// TIA Portal V20 program export: 7 tag tables, 9 data types, 98 data blocks, 45 code blocks (in call order from the OBs), 102 instance data blocks

VAR_GLOBAL   // PLC tag table "00_Simulation"
   "AAxxxSP1.Slot1.I.16" AT %I1.0 : Bool;   // SIMIT Simulation currently running (life bit from SIMIT, always TRUE while SIMIT is running)
END_VAR

VAR_GLOBAL   // PLC tag table "06_ProductionData"
END_VAR
VAR_GLOBAL CONSTANT   // user constants
   NO_DATASETS_CYCLETIMER : Int := 8;   // SICAR: Anzahl Datensätze Taktzeiten / SICAR: Number of data sets Cycle Timer
   NO_DATASETS_LIMITVALUES : Int := 2;   // SICAR: Anzahl Datensätze Grenzwerte / SICAR: Number of data sets Limit Value
   NO_DATASETS_SHIFTCOUNTER : Int := 2;   // SICAR: Anzahl Datensätze Schichtzähler / SICAR: Number of data sets Shift Counter
   NO_DATASETS_COUNTER : Int := 2;   // SICAR: Anzahl Datensätze Zähler / SICAR: Number of data sets Counter
END_VAR

VAR_GLOBAL   // PLC tag table "07_Energy"
   PAC3220InPut AT %I500.0 : "LER_typePAC3220ProfinetInput";
   PAC3220OutPut AT %Q500.0 : "LER_typePAC3220ProfinetOutput";
   "Active energy import tariff 1(F)" AT %ID612 : Real;
   "Reactive energy import tariff 1 (F)" AT %ID616 : Real;
   "Apparent energy tariff 1 (F)" AT %ID620 : Real;
   "Active energy export tariff 1(F)" AT %ID624 : Real;
   "Reactive energy export tariff 1 (F)" AT %ID628 : Real;
   "Apparent power L1" AT %ID632 : Real;
   "Apparent power L2" AT %ID636 : Real;
   "Apparent power L3" AT %ID640 : Real;
   "Active power L1" AT %ID644 : Real;
   "Active power L2" AT %ID648 : Real;
   "Active power L3" AT %ID652 : Real;
   "Reactive power L1" AT %ID656 : Real;
   "Reactive power L2" AT %ID660 : Real;
   "Reactive power L3" AT %ID664 : Real;
END_VAR
VAR_GLOBAL CONSTANT   // user constants
   NO_OF_MACHINES : USInt := 1;   // SICAR: No of machines for EE-Monitor
   NO_OF_MEASUREPOINTS : USInt := 1;   // SICAR: Anzahl der Messstellen für EE-Monitor / SICAR: No of measurepoints for EE-Monitor
   "DP_FRWA1_1_0_000CC1-KE50~DP_FRWA1_1_0_000CC1-KE50_900" : Hw_Io := 577;
END_VAR

VAR_GLOBAL   // PLC tag table "08_CmInfo"
END_VAR
VAR_GLOBAL CONSTANT   // user constants
   NO_OF_RF_IDENT_DEVICES : USInt := 1;   // SICAR: Anzahl der RF Lesestellen / SICAR: Number of RF readers
   NO_OF_MV_IDENT_DEVICES : USInt := 1;   // SICAR: Anzahl der MV Lesestellen / SICAR: Number of MV readers
   NO_OF_ET200SPMOTORSTARTER : USInt := 1;   // SICAR: Anzahl Motorstarter / SICAR: Number of ET200SP Motorstarter
END_VAR

VAR_GLOBAL   // PLC tag table "11_Settings"
END_VAR
VAR_GLOBAL CONSTANT   // user constants
   MAX_NO_OF_DEVICES_X1 : Int := 200;
   MAX_NO_OF_MODULES_X1 : Int := 200;
   MAX_NO_OF_DEVICES_X2 : Int := 200;
   MAX_NO_OF_MODULES_X2 : Int := 200;
END_VAR

VAR_GLOBAL   // PLC tag table "CentralFunctions"
END_VAR

VAR_GLOBAL   // PLC tag table "TextListId"
END_VAR
VAR_GLOBAL CONSTANT   // user constants
   TEXT_LIST_ID_PN_DEV_DIAG : Int := 591;   // SICAR: ID von SPS Alarm Textlist / SICAR: ID of PLC Alarm text list
   TEXT_LIST_ID_CHECKSUM : Int := 584;   // SICAR: ID von SPS Alarm Textlist / SICAR: ID of PLC Alarm text list
   TEXT_LIST_ID_EEEMONITOR_REPORT : Int := 562;   // SICAR: ID von SPS Alarm Textlist / SICAR: ID of PLC Alarm text list
   TEXT_LIST_ID_EEEMONITOR_CALC : Int := 561;   // SICAR: ID von SPS Alarm Textlist / SICAR: ID of PLC Alarm text list
   TEXT_LIST_ID_IDENT_SYSTEM : Int := 516;   // SICAR: ID of PLC Alarm for ident demo
   TEXT_LIST_ID_SMC_PD : Int := 585;   // SICAR: ID von SPS Alarm Textlist / SICAR: ID of PLC Alarm text list
   TEXT_LIST_ID_MOTORSTARTERS : Int := 588;   // SICAR: ID of PLC Alarm for motorstarter Demo
   TEXT_LIST_ID_DEV_FWD_REV : Int := 592;   // SICAR: ID of PLC Alarm for motorstarter Demo
END_VAR

TYPE "typeReelCutToStack"
   STRUCT
      Load_Enable : Bool;
      Load_Complete_Comfirm : Bool;
      Cell_Data_Report : Bool;
      signal3 : Bool;
      signal4 : Bool;
      signal5 : Bool;
      signal6 : Bool;
      signal7 : Bool;
      signal8 : Bool;
      signal9 : Bool;
      signal10 : Bool;
      signal11 : Bool;
      signal12 : Bool;
      signal13 : Bool;
      signal14 : Bool;
      HeartBeat : Bool;
      signal16 : Bool;
      signal17 : Bool;
      signal18 : Bool;
      signal19 : Bool;
      signal20 : Bool;
      signal21 : Bool;
      signal22 : Bool;
      signal23 : Bool;
      signal24 : Bool;
      signal25 : Bool;
      signal26 : Bool;
      signal27 : Bool;
      signal28 : Bool;
      signal29 : Bool;
      signal30 : Bool;
      signal31 : Bool;
      signal32 : Bool;
      signal33 : Bool;
      signal34 : Bool;
      signal35 : Bool;
      signal36 : Bool;
      signal37 : Bool;
      signal38 : Bool;
      signal39 : Bool;
      signal40 : Bool;
      signal41 : Bool;
      signal42 : Bool;
      signal43 : Bool;
      signal44 : Bool;
      signal45 : Bool;
      signal46 : Bool;
      signal47 : Bool;
      signal48 : Bool;
      signal49 : Bool;
      signal50 : Bool;
      signal51 : Bool;
      signal52 : Bool;
      signal53 : Bool;
      signal54 : Bool;
      signal55 : Bool;
      signal56 : Bool;
      signal57 : Bool;
      signal58 : Bool;
      signal59 : Bool;
      signal60 : Bool;
      signal61 : Bool;
      signal62 : Bool;
      signal63 : Bool;
      signal64 : Bool;
      signal65 : Bool;
      signal66 : Bool;
      signal67 : Bool;
      signal68 : Bool;
      signal69 : Bool;
      signal70 : Bool;
      signal71 : Bool;
      signal72 : Bool;
      signal73 : Bool;
      signal74 : Bool;
      signal75 : Bool;
      signal76 : Bool;
      signal77 : Bool;
      signal78 : Bool;
      signal79 : Bool;
      signal80 : Bool;
      signal81 : Bool;
      signal82 : Bool;
      signal83 : Bool;
      signal84 : Bool;
      signal85 : Bool;
      signal86 : Bool;
      signal87 : Bool;
      signal88 : Bool;
      signal89 : Bool;
      signal90 : Bool;
      signal91 : Bool;
      signal92 : Bool;
      signal93 : Bool;
      signal94 : Bool;
      signal95 : Bool;
   END_STRUCT;
END_TYPE

TYPE "typeStackToReelCut"
   STRUCT
      Load_Requset : Bool;
      Load_Busy : Bool;
      Load_Complete : Bool;
      Cell_Data_Request : Bool;
      Cell_Data_Report_Ack : Bool;
      Cell_Data_Report_Nck : Bool;
      signal6 : Bool;
      signal7 : Bool;
      signal8 : Bool;
      signal9 : Bool;
      signal10 : Bool;
      signal11 : Bool;
      signal12 : Bool;
      signal13 : Bool;
      signal14 : Bool;
      HeartBeat : Bool;
      signal16 : Bool;
      signal17 : Bool;
      signal18 : Bool;
      signal19 : Bool;
      signal20 : Bool;
      signal21 : Bool;
      signal22 : Bool;
      signal23 : Bool;
      signal24 : Bool;
      signal25 : Bool;
      signal26 : Bool;
      signal27 : Bool;
      signal28 : Bool;
      signal29 : Bool;
      signal30 : Bool;
      signal31 : Bool;
      signal32 : Bool;
      signal33 : Bool;
      signal34 : Bool;
      signal35 : Bool;
      signal36 : Bool;
      signal37 : Bool;
      signal38 : Bool;
      signal39 : Bool;
      signal40 : Bool;
      signal41 : Bool;
      signal42 : Bool;
      signal43 : Bool;
      signal44 : Bool;
      signal45 : Bool;
      signal46 : Bool;
      signal47 : Bool;
      signal48 : Bool;
      signal49 : Bool;
      signal50 : Bool;
      signal51 : Bool;
      signal52 : Bool;
      signal53 : Bool;
      signal54 : Bool;
      signal55 : Bool;
      signal56 : Bool;
      signal57 : Bool;
      signal58 : Bool;
      signal59 : Bool;
      signal60 : Bool;
      signal61 : Bool;
      signal62 : Bool;
      signal63 : Bool;
      signal64 : Bool;
      signal65 : Bool;
      signal66 : Bool;
      signal67 : Bool;
      signal68 : Bool;
      signal69 : Bool;
      signal70 : Bool;
      signal71 : Bool;
      signal72 : Bool;
      signal73 : Bool;
      signal74 : Bool;
      signal75 : Bool;
      signal76 : Bool;
      signal77 : Bool;
      signal78 : Bool;
      signal79 : Bool;
      signal80 : Bool;
      signal81 : Bool;
      signal82 : Bool;
      signal83 : Bool;
      signal84 : Bool;
      signal85 : Bool;
      signal86 : Bool;
      signal87 : Bool;
      signal88 : Bool;
      signal89 : Bool;
      signal90 : Bool;
      signal91 : Bool;
      signal92 : Bool;
      signal93 : Bool;
      signal94 : Bool;
      signal95 : Bool;
   END_STRUCT;
END_TYPE

TYPE "typeEmMotorStarterInterface"
// stored: Access Published
   STRUCT
      EMmotorstarter : Array[0.."NO_OF_EM"] of "typeMotorStarterInterface";
   END_STRUCT;
END_TYPE

TYPE "typeEt200SpMotorstarterInterfaceHmi"
// stored: Access Published
   STRUCT
      et200SpMotorstarterReadValue : Bool;   // read Value of MotorStarter
      et200SpNumberOfMotorstarters { ExternalWritable := 'False'} : USInt;   // Number of Motor Starters
      et200SpUnitMotorstarter : USInt := 1;   // Unit selected
      et200SpEMMotorstarter : USInt := 0;   // Equipment Module selected
      et200SpMotorstarterCurrent : Array[0.."NO_OF_ET200SPMOTORSTARTER"] of Real;   // Aktuelle Werte / Current values
      et200SpMotorstarterInputs : Array[0.."NO_OF_ET200SPMOTORSTARTER"] of "LSicar_typeMotorstarterIn";   // Motorstarter Data Inputs HMI
      et200SpMotorstarterOutputs : Array[0.."NO_OF_ET200SPMOTORSTARTER"] of "LSicar_typeMotorstarterOut";   // Motorstarter Data Outputs HMI
   END_STRUCT;
END_TYPE

TYPE "typeMotorStarterInterface"
// stored: Access Published
   STRUCT
      et200SpMotorstarterCurrent : Array[0.."NO_OF_ET200SPMOTORSTARTER"] of Real;   // Aktuelle Werte / Current values
      et200SpMotorstarterInputs : Array[0.."NO_OF_ET200SPMOTORSTARTER"] of "LSicar_typeMotorstarterIn";   // Motorstarter Data Inputs HMI
      et200SpMotorstarterOutputs : Array[0.."NO_OF_ET200SPMOTORSTARTER"] of "LSicar_typeMotorstarterOut";   // Motorstarter Data Outputs HMI
   END_STRUCT;
END_TYPE

TYPE "typeEMIdentMv"
// stored: Access Published
   STRUCT
      identMvEM : Array[0.."NO_OF_EM"] of "typeIdentMvHmi";
   END_STRUCT;
END_TYPE

TYPE "typeIdentMvHmi"
// stored: Access Published
   STRUCT
      selectedUnit : USInt;
      selectedEM : USInt;
      mvReaderId : USInt;   // MV Reader ID
      numberOfMv : USInt;   // Anzahl der MV Antriebe / Number of used MV readers
      mvReader : Array[0.."NO_OF_MV_IDENT_DEVICES"] of "LSicar_typeIdentInterfaceHmi";   // MV Reader
   END_STRUCT;
END_TYPE

TYPE "typeEMIdentRf"
// stored: Access Published
   STRUCT
      identRfEM : Array[0.."NO_OF_EM"] of "typeIdentRfHmi";
   END_STRUCT;
END_TYPE

TYPE "typeIdentRfHmi"
// stored: Access Published
   STRUCT
      selectedUnit : USInt;
      selectedEM : USInt;
      rfReaderId : USInt;   // Reader ID / RF Reader ID
      numberOfRf : USInt;   // Anzahl der RFID Antriebe / Number of used RFIDs
      rfReader : Array[0.."NO_OF_RF_IDENT_DEVICES"] of "LSicar_typeIdentInterfaceHmi";   // RF Reader
   END_STRUCT;
END_TYPE

DATA_BLOCK "TestTemp"   // DB503
// stored: MemoryReserve 100
   VAR
      TempBool : Array[0..100] of Bool;
   END_VAR
BEGIN
END_DATA_BLOCK

DATA_BLOCK "Hmi"   // DB4
// stored: MemoryReserve 100
   VAR
      mainHeader : Array[0.."NO_OF_PANELS"] of "LAF_typeHeader";   // Input from the status bar of the HMI
      operationInterlock : "LAF_typeOperationInterlockInterface";
      TestBit { S7_SetPoint := 'True'} : Array[0..9] of Bool;
   END_VAR
BEGIN
   mainHeader[0..1].hmiToPlc.acknowledge := FALSE;
   mainHeader[0..1].hmiToPlc.powerCommands := 16#00;
   mainHeader[0..1].hmiToPlc.selectedUnits := 16#0001;
   mainHeader[0..1].hmiToPlc.modeRequests := 16#0000;
   mainHeader[0..1].hmiToPlc.stateCommands := 16#0000;
   mainHeader[0..1].hmiToPlc.specialFunctions := 16#0000;
   mainHeader[0..1].plcToHmi.powerStatus := 0;
   mainHeader[0..1].plcToHmi.displayedMode := 2;
   mainHeader[0..1].plcToHmi.displayedState := 2;
   mainHeader[0..1].plcToHmi.modeRequestsButtons.visibility := 16#000F;
   mainHeader[0].plcToHmi.modeRequestsButtons.operatorControlAllowed := 16#000F;
   mainHeader[1].plcToHmi.modeRequestsButtons.operatorControlAllowed := 16#0001;
   mainHeader[0..1].plcToHmi.modeRequestsButtons.active := 16#0002;
   mainHeader[0].plcToHmi.stateCommandsButtons.visibility := 16#0000;
   mainHeader[1].plcToHmi.stateCommandsButtons.visibility := 16#000F;
   mainHeader[0..1].plcToHmi.stateCommandsButtons.operatorControlAllowed := 16#0084;
   mainHeader[0..1].plcToHmi.stateCommandsButtons.active := 16#0000;
   mainHeader[0].plcToHmi.specialFunctionButtons.visibility := 16#701fffff;
   mainHeader[1].plcToHmi.specialFunctionButtons.visibility := 16#0007;
   mainHeader[0].plcToHmi.specialFunctionButtons.operatorControlAllowed := 16#701fffff;
   mainHeader[1].plcToHmi.specialFunctionButtons.operatorControlAllowed := 16#000F;
   mainHeader[0..1].plcToHmi.specialFunctionButtons.active := 16#0000;
   operationInterlock.commands.reqMaintenanceLock := FALSE;
   operationInterlock.commands.reqMaintenanceReset := FALSE;
   operationInterlock.commands.serverMachineName := WSTRING#'ucp-3013893F1460';
   operationInterlock.commands.localMachineName := WSTRING#'Controlroom Client';
   operationInterlock.monitoring.maintenanceLockActive := FALSE;
END_DATA_BLOCK

DATA_BLOCK "LRemoteAccess_Data"   // DB275
TITLE = Data
AUTHOR : Siemens
// Storing data about mobile panel and UCP connection status
// stored: Access Published, MemoryReserve 100
   VAR
      mobilePanel1 : "LRemoteAccess_typeMobilePanel";
      connectionBoxes : Array[1..2] of "LRemoteAccess_typeConnectionBox";
      ActivationMobileDP { S7_SetPoint := 'True'} : "LRemoteAccess_typeMobile_DeActivate";   // Activate Mobile Panel
      DeactivationMobileDP { S7_SetPoint := 'True'} : "LRemoteAccess_typeMobile_DeActivate";   // Deactivate Mobile Panel
      connectionTimeout { S7_SetPoint := 'True'} : Time := T#5S;   // Connection timeout. Keep greater than 3 sec. Default 5 sec.
   END_VAR
BEGIN
   mobilePanel1.connectionTerminated := FALSE;
   mobilePanel1.mpReadBoxID := 0;
   mobilePanel1.mpLifeBit := 5;
   mobilePanel1.mpDesignator := WSTRING#'';
   mobilePanel1.mpKeySwitch := 0;
   mobilePanel1.ucpPointerEnabled := TRUE;
   mobilePanel1.ucpPointerDisabled := FALSE;
   connectionBoxes[1].ID := 18;
   connectionBoxes[2].ID := 19;
   connectionBoxes[1..2].connected := FALSE;
   ActivationMobileDP.Execute := FALSE;
   ActivationMobileDP.RET_VAL := 28672;
   ActivationMobileDP.Busy := FALSE;
   DeactivationMobileDP.Execute := FALSE;
   DeactivationMobileDP.RET_VAL := 28672;
   DeactivationMobileDP.Busy := FALSE;
END_DATA_BLOCK

DATA_BLOCK "Simulation"   // DB203
TITLE = Simulation
// Simulation data
// stored: MemoryReserve 100
   VAR
      simHmiRotaryAxis : Array[0..49] of "LER_typeSimRotaryAxis";
      simHmiLinearAxis : Array[0..49] of "LER_typeSimLinearAxis";
      data : "LAF_typeSimulation";
   END_VAR
BEGIN
   data.simitActive := FALSE;
   data.simulationActiveHmi := FALSE;
   data.showSimulationButtonHmi := TRUE;
END_DATA_BLOCK

DATA_BLOCK "HMI_Interface_Overview"   // DB276
// stored: Access Published, MemoryReserve 100
   VAR
      State : Struct
         "Anode Reel Cut" : "HMI_IF_OverView_Unit_UDT";
         "Cathode Reel Cut" : "HMI_IF_OverView_Unit_UDT";
         "Stacker #1" : "HMI_IF_OverView_Unit_UDT";
         "Stacker #2" : "HMI_IF_OverView_Unit_UDT";
         Inspection : "HMI_IF_OverView_Unit_UDT";
      END_STRUCT;
   END_VAR
BEGIN
   State."Anode Reel Cut".State.Communication := 0;
   State."Anode Reel Cut".State.Mode := 0;
   State."Anode Reel Cut".State.State := 0;
   State."Anode Reel Cut".State.Emergency := 0;
   State."Anode Reel Cut"."Link&Unlink".Em0 := FALSE;
   State."Anode Reel Cut"."Link&Unlink".Em1 := FALSE;
   State."Anode Reel Cut"."Link&Unlink".Em2 := FALSE;
   State."Anode Reel Cut"."Link&Unlink".Em3 := FALSE;
   State."Anode Reel Cut"."Link&Unlink".Em4 := FALSE;
   State."Anode Reel Cut"."Link&Unlink".Em5 := FALSE;
   State."Anode Reel Cut"."Link&Unlink".Em6 := FALSE;
   State."Anode Reel Cut"."Link&Unlink".Em7 := FALSE;
   State."Anode Reel Cut"."Link&Unlink".Em8 := FALSE;
   State."Anode Reel Cut"."Link&Unlink".Em9 := FALSE;
   State."Anode Reel Cut"."Link&Unlink".Em10 := FALSE;
   State."Anode Reel Cut"."Link&Unlink".Em11 := FALSE;
   State."Anode Reel Cut"."Link&Unlink".Em12 := FALSE;
   State."Anode Reel Cut"."Link&Unlink".Em13 := FALSE;
   State."Anode Reel Cut"."Link&Unlink".Em14 := FALSE;
   State."Anode Reel Cut"."Link&Unlink".Em15 := FALSE;
   State."Anode Reel Cut".Production."Total Input Quantity" := 0;
   State."Anode Reel Cut".Production."Remain Count" := 0;
   State."Anode Reel Cut".Production."Processed Count" := 0;
   State."Anode Reel Cut".Production."NG Count" := 0;
   State."Cathode Reel Cut".State.Communication := 0;
   State."Cathode Reel Cut".State.Mode := 0;
   State."Cathode Reel Cut".State.State := 0;
   State."Cathode Reel Cut".State.Emergency := 0;
   State."Cathode Reel Cut"."Link&Unlink".Em0 := FALSE;
   State."Cathode Reel Cut"."Link&Unlink".Em1 := FALSE;
   State."Cathode Reel Cut"."Link&Unlink".Em2 := FALSE;
   State."Cathode Reel Cut"."Link&Unlink".Em3 := FALSE;
   State."Cathode Reel Cut"."Link&Unlink".Em4 := FALSE;
   State."Cathode Reel Cut"."Link&Unlink".Em5 := FALSE;
   State."Cathode Reel Cut"."Link&Unlink".Em6 := FALSE;
   State."Cathode Reel Cut"."Link&Unlink".Em7 := FALSE;
   State."Cathode Reel Cut"."Link&Unlink".Em8 := FALSE;
   State."Cathode Reel Cut"."Link&Unlink".Em9 := FALSE;
   State."Cathode Reel Cut"."Link&Unlink".Em10 := FALSE;
   State."Cathode Reel Cut"."Link&Unlink".Em11 := FALSE;
   State."Cathode Reel Cut"."Link&Unlink".Em12 := FALSE;
   State."Cathode Reel Cut"."Link&Unlink".Em13 := FALSE;
   State."Cathode Reel Cut"."Link&Unlink".Em14 := FALSE;
   State."Cathode Reel Cut"."Link&Unlink".Em15 := FALSE;
   State."Cathode Reel Cut".Production."Total Input Quantity" := 0;
   State."Cathode Reel Cut".Production."Remain Count" := 0;
   State."Cathode Reel Cut".Production."Processed Count" := 0;
   State."Cathode Reel Cut".Production."NG Count" := 0;
   State."Stacker #1".State.Communication := 0;
   State."Stacker #1".State.Mode := 0;
   State."Stacker #1".State.State := 0;
   State."Stacker #1".State.Emergency := 0;
   State."Stacker #1"."Link&Unlink".Em0 := FALSE;
   State."Stacker #1"."Link&Unlink".Em1 := FALSE;
   State."Stacker #1"."Link&Unlink".Em2 := FALSE;
   State."Stacker #1"."Link&Unlink".Em3 := FALSE;
   State."Stacker #1"."Link&Unlink".Em4 := FALSE;
   State."Stacker #1"."Link&Unlink".Em5 := FALSE;
   State."Stacker #1"."Link&Unlink".Em6 := FALSE;
   State."Stacker #1"."Link&Unlink".Em7 := FALSE;
   State."Stacker #1"."Link&Unlink".Em8 := FALSE;
   State."Stacker #1"."Link&Unlink".Em9 := FALSE;
   State."Stacker #1"."Link&Unlink".Em10 := FALSE;
   State."Stacker #1"."Link&Unlink".Em11 := FALSE;
   State."Stacker #1"."Link&Unlink".Em12 := FALSE;
   State."Stacker #1"."Link&Unlink".Em13 := FALSE;
   State."Stacker #1"."Link&Unlink".Em14 := FALSE;
   State."Stacker #1"."Link&Unlink".Em15 := FALSE;
   State."Stacker #1".Production."Total Input Quantity" := 0;
   State."Stacker #1".Production."Remain Count" := 0;
   State."Stacker #1".Production."Processed Count" := 0;
   State."Stacker #1".Production."NG Count" := 0;
   State."Stacker #2".State.Communication := 0;
   State."Stacker #2".State.Mode := 0;
   State."Stacker #2".State.State := 0;
   State."Stacker #2".State.Emergency := 0;
   State."Stacker #2"."Link&Unlink".Em0 := FALSE;
   State."Stacker #2"."Link&Unlink".Em1 := FALSE;
   State."Stacker #2"."Link&Unlink".Em2 := FALSE;
   State."Stacker #2"."Link&Unlink".Em3 := FALSE;
   State."Stacker #2"."Link&Unlink".Em4 := FALSE;
   State."Stacker #2"."Link&Unlink".Em5 := FALSE;
   State."Stacker #2"."Link&Unlink".Em6 := FALSE;
   State."Stacker #2"."Link&Unlink".Em7 := FALSE;
   State."Stacker #2"."Link&Unlink".Em8 := FALSE;
   State."Stacker #2"."Link&Unlink".Em9 := FALSE;
   State."Stacker #2"."Link&Unlink".Em10 := FALSE;
   State."Stacker #2"."Link&Unlink".Em11 := FALSE;
   State."Stacker #2"."Link&Unlink".Em12 := FALSE;
   State."Stacker #2"."Link&Unlink".Em13 := FALSE;
   State."Stacker #2"."Link&Unlink".Em14 := FALSE;
   State."Stacker #2"."Link&Unlink".Em15 := FALSE;
   State."Stacker #2".Production."Total Input Quantity" := 0;
   State."Stacker #2".Production."Remain Count" := 0;
   State."Stacker #2".Production."Processed Count" := 0;
   State."Stacker #2".Production."NG Count" := 0;
   State.Inspection.State.Communication := 0;
   State.Inspection.State.Mode := 0;
   State.Inspection.State.State := 0;
   State.Inspection.State.Emergency := 0;
   State.Inspection."Link&Unlink".Em0 := FALSE;
   State.Inspection."Link&Unlink".Em1 := FALSE;
   State.Inspection."Link&Unlink".Em2 := FALSE;
   State.Inspection."Link&Unlink".Em3 := FALSE;
   State.Inspection."Link&Unlink".Em4 := FALSE;
   State.Inspection."Link&Unlink".Em5 := FALSE;
   State.Inspection."Link&Unlink".Em6 := FALSE;
   State.Inspection."Link&Unlink".Em7 := FALSE;
   State.Inspection."Link&Unlink".Em8 := FALSE;
   State.Inspection."Link&Unlink".Em9 := FALSE;
   State.Inspection."Link&Unlink".Em10 := FALSE;
   State.Inspection."Link&Unlink".Em11 := FALSE;
   State.Inspection."Link&Unlink".Em12 := FALSE;
   State.Inspection."Link&Unlink".Em13 := FALSE;
   State.Inspection."Link&Unlink".Em14 := FALSE;
   State.Inspection."Link&Unlink".Em15 := FALSE;
   State.Inspection.Production."Total Input Quantity" := 0;
   State.Inspection.Production."Remain Count" := 0;
   State.Inspection.Production."Processed Count" := 0;
   State.Inspection.Production."NG Count" := 0;
END_DATA_BLOCK

DATA_BLOCK "LAF_InternalManual"   // DB43
VERSION : 19.0
// stored: MemoryReserve 100
   VAR
      hmi : Array[1..1] of "LAF_typeManHmiDisp";   // Anzahl der HMIs - modifizieren Sie die Array-Größe auf Basis der erforderlichen HMI / number of HMIs - modify the array size based on the required HMIs / número de HMI: modificar el tamaño del array según las HMI requeridas / nombre d'IHM - modifier la taille du tableau en fonction du nombre d'IHM requis / numero di HMI - modificare la dimensione di array in base alle HMI richieste / HMI 수 - 필요한 HMI에 따라 배열 크기를 수정합니다. / HMI 数量 - 根据所需的 HMI 修改数组大小
      manualOperationEnabled : Bool;   // feedback whether the manual operation lines are selected
      emsWithManualOpConfigured { ExternalWritable := 'False'} : "LGM_emsWithManualOpConfigured";   // List of EMs with manual operation configured, for HMI button visibility
      disableUnit1 { S7_SetPoint := 'True'} : Bool;
      RisingEdge : Bool;
   END_VAR
BEGIN
END_DATA_BLOCK

DATA_BLOCK "OperatorPrompts"   // DB123
// stored: Access Published, MemoryReserve 100
   VAR
      triggers { ExternalAccessible := 'False'; ExternalVisible := 'False'; ExternalWritable := 'False'} : Array[1..63] of Bool;
      activeOperatorPrompt { ExternalWritable := 'False'} : Int := 0;
      ack : Bool := FALSE;
   END_VAR
BEGIN
   triggers[1..63] := FALSE;
END_DATA_BLOCK

DATA_BLOCK "ProdDataInterfaceHmi"   // DB53
TITLE = HMI und Anwender Schnittstelle für Produktionsdaten / HMI and user interface for production data
AUTHOR : SICAR
FAMILY : ProdData
// FUNKTIONSBESCHREIBUNG: 
// Der Baustein beinhaltet alle Informationen zum und vom HMI, sowie die Anwenderschnittstellen für die Produktionsdaten
// Weitere Hinweise: siehe SICAR anwenderdefinierte Dokumentation / SICAR Online-Hilfe.
// DESCRIPTION OF FUNCTIONS:
// stored: MemoryReserve 100
   VAR RETAIN
      numberOfDataSets : "LSicar_typeNumberOfDataSets";   // Anzahl konfigurierter Datensätze / Number of configured data sets
   END_VAR
   VAR
      colorCodeLimitSummary : UInt := 0;   // Gesamt Status Grenzwerte / Overall status Limit values
      colorCodeLimitSelButton : Array[0..8] of UInt;   // Farbcode für Datensatz Anwahl Button (Grenzwerte) / Color code for data set select button (Limit values)
   END_VAR
   VAR RETAIN
      limitValueDataSetSel : Int := 1;   // Angwaehlter Datensatz Grenzwerte / selected data set limit values
      limitDataSet : Array[0.."NO_DATASETS_LIMITVALUES"] of "LSicar_typeLimitValue";   // Datensätze Grenzwerte / Data sets limit .values
      cycleTimerDataSetSel : Int := 1;   // Angewaehlter Datensatz Taktzeiten / selected data set cycle timer
      cycleTimerDataSet : Array[0.."NO_DATASETS_CYCLETIMER"] of "LSicar_typeCycleTimer";   // Datensätze Taktzeiten / Data sets cycle timer
      counterDataSetSel : Int := 1;   // Angewählter Datensatz Zaehler / selected data set counter
      counterDataSet : Array[0.."NO_DATASETS_COUNTER"] of "LSicar_typeCounter";   // Datensätze Zähler / Data sets counter
      shiftCounterDataSetSel : Int := 1;   // Angewaehlter Datensatz Schichtzaehler / selected data set shift counter
      shiftCounterDataSet : Array[0.."NO_DATASETS_SHIFTCOUNTER"] of "LSicar_typeShiftCounter";   // Datensätze Schichtzähler / Data sets shift counter
      shiftCountOeeDataSetSel : Int := 1;   // Angewaehlter Datensatz OEE / selected data set OEE
      shiftCounterOeeDataSet : Array[0.."NO_DATASETS_SHIFTCOUNTER"] of "LSicar_typeShiftCounterOee";   // Datensätze Schichtzähler OEE / Data sets shift counter OEE
   END_VAR
BEGIN
   numberOfDataSets.limitValues := 2;
   numberOfDataSets.cycleTimer := 2;
   numberOfDataSets."counter" := 2;
   numberOfDataSets.shiftCounter := 2;
   colorCodeLimitSelButton[0..8] := 0;
   limitDataSet[0].targetValue[0..10] := 0;
   limitDataSet[1].targetValue[0..10] := 0;
   limitDataSet[2].targetValue[0..10] := 0;
   limitDataSet[0].prewarnValue[0..10] := 0;
   limitDataSet[1].prewarnValue[0..10] := 0;
   limitDataSet[2].prewarnValue[0..10] := 0;
   limitDataSet[0].remainValue[0..10] := 0;
   limitDataSet[1].remainValue[0..10] := 0;
   limitDataSet[2].remainValue[0..10] := 0;
   limitDataSet[0].control[0..10].count := FALSE;
   limitDataSet[1].control[0..10].count := FALSE;
   limitDataSet[2].control[0..10].count := FALSE;
   limitDataSet[0].control[0..10].set := FALSE;
   limitDataSet[1].control[0..10].set := FALSE;
   limitDataSet[2].control[0..10].set := FALSE;
   limitDataSet[0].control[0..10].prewarn := FALSE;
   limitDataSet[1].control[0..10].prewarn := FALSE;
   limitDataSet[2].control[0..10].prewarn := FALSE;
   limitDataSet[0].control[0..10].alarm := FALSE;
   limitDataSet[1].control[0..10].alarm := FALSE;
   limitDataSet[2].control[0..10].alarm := FALSE;
   limitDataSet[0].textListValue[0..10] := 0;
   limitDataSet[1].textListValue[0..10] := 0;
   limitDataSet[2].textListValue[0..10] := 0;
   limitDataSet[0..2].userInterfaceVisibility := 16#0000_0000;
   limitDataSet[0].colorCodeAlarmPrewarn[0..10] := 0;
   limitDataSet[1].colorCodeAlarmPrewarn[0..10] := 0;
   limitDataSet[2].colorCodeAlarmPrewarn[0..10] := 0;
   limitDataSet[0..2].indexSelectedLimitValue := 0;
   limitDataSet[0..2].divButton := 16#00;
   limitDataSet[0..2].visibility := 16#0000_0000;
   cycleTimerDataSet[0].targetValue[0..20] := 0;
   cycleTimerDataSet[1].targetValue[0..20] := 0;
   cycleTimerDataSet[2].targetValue[0..20] := 0;
   cycleTimerDataSet[0].currentValue[0..20] := 0;
   cycleTimerDataSet[1].currentValue[0..20] := 0;
   cycleTimerDataSet[2].currentValue[0..20] := 0;
   cycleTimerDataSet[0].averageValue[0..20] := 0;
   cycleTimerDataSet[1].averageValue[0..20] := 0;
   cycleTimerDataSet[2].averageValue[0..20] := 0;
   cycleTimerDataSet[0].counts[0..20] := 0;
   cycleTimerDataSet[1].counts[0..20] := 0;
   cycleTimerDataSet[2].counts[0..20] := 0;
   cycleTimerDataSet[0].measureActive[0..20] := 0;
   cycleTimerDataSet[1].measureActive[0..20] := 0;
   cycleTimerDataSet[2].measureActive[0..20] := 0;
   cycleTimerDataSet[0].control[0..20].run := FALSE;
   cycleTimerDataSet[1].control[0..20].run := FALSE;
   cycleTimerDataSet[2].control[0..20].run := FALSE;
   cycleTimerDataSet[0].control[0..20].hold := FALSE;
   cycleTimerDataSet[1].control[0..20].hold := FALSE;
   cycleTimerDataSet[2].control[0..20].hold := FALSE;
   cycleTimerDataSet[0].control[0..20].reset := FALSE;
   cycleTimerDataSet[1].control[0..20].reset := FALSE;
   cycleTimerDataSet[2].control[0..20].reset := FALSE;
   cycleTimerDataSet[0].textListValue[0..20] := 0;
   cycleTimerDataSet[1].textListValue[0..20] := 0;
   cycleTimerDataSet[2].textListValue[0..20] := 0;
   cycleTimerDataSet[0..2].userInterfaceVisibility := 16#0000_0000;
   cycleTimerDataSet[0..2].resetAverageAllExt := FALSE;
   cycleTimerDataSet[0..2].indexSelectedTimer := 0;
   cycleTimerDataSet[0..2].divButton := 16#00;
   cycleTimerDataSet[0..2].visibility := 16#0000_0000;
   counterDataSet[0].currentValue[0..20] := 0;
   counterDataSet[1].currentValue[0..20] := 0;
   counterDataSet[2].currentValue[0..20] := 0;
   counterDataSet[0].control[0..20].countUp := FALSE;
   counterDataSet[1].control[0..20].countUp := FALSE;
   counterDataSet[2].control[0..20].countUp := FALSE;
   counterDataSet[0].control[0..20].countDown := FALSE;
   counterDataSet[1].control[0..20].countDown := FALSE;
   counterDataSet[2].control[0..20].countDown := FALSE;
   counterDataSet[0].control[0..20].reset := FALSE;
   counterDataSet[1].control[0..20].reset := FALSE;
   counterDataSet[2].control[0..20].reset := FALSE;
   counterDataSet[0].textListValue[0..20] := 0;
   counterDataSet[1].textListValue[0..20] := 0;
   counterDataSet[2].textListValue[0..20] := 0;
   counterDataSet[0].userInterfaceVisibility := 16#0000_0000;
   counterDataSet[1].userInterfaceVisibility := 16#0000_0007;
   counterDataSet[2].userInterfaceVisibility := 16#0000_0003;
   counterDataSet[0..2].resetAllExt := FALSE;
   counterDataSet[0..2].indexSelectedCounter := 0;
   counterDataSet[0..2].divButton := 16#00;
   counterDataSet[0..2].visibility := 16#0000_0000;
   shiftCounterDataSet[0].currentShiftValue.partsTarget[0..10] := 0;
   shiftCounterDataSet[1].currentShiftValue.partsTarget[0..10] := 0;
   shiftCounterDataSet[2].currentShiftValue.partsTarget[0..10] := 0;
   shiftCounterDataSet[0].currentShiftValue.partsCurrent[0..10] := 0;
   shiftCounterDataSet[1].currentShiftValue.partsCurrent[0..10] := 0;
   shiftCounterDataSet[2].currentShiftValue.partsCurrent[0..10] := 0;
   shiftCounterDataSet[0].previousShiftValue.partsTarget[0..10] := 0;
   shiftCounterDataSet[1].previousShiftValue.partsTarget[0..10] := 0;
   shiftCounterDataSet[2].previousShiftValue.partsTarget[0..10] := 0;
   shiftCounterDataSet[0].previousShiftValue.partsCurrent[0..10] := 0;
   shiftCounterDataSet[1].previousShiftValue.partsCurrent[0..10] := 0;
   shiftCounterDataSet[2].previousShiftValue.partsCurrent[0..10] := 0;
   shiftCounterDataSet[0].penultimateShiftValue.partsTarget[0..10] := 0;
   shiftCounterDataSet[1].penultimateShiftValue.partsTarget[0..10] := 0;
   shiftCounterDataSet[2].penultimateShiftValue.partsTarget[0..10] := 0;
   shiftCounterDataSet[0].penultimateShiftValue.partsCurrent[0..10] := 0;
   shiftCounterDataSet[1].penultimateShiftValue.partsCurrent[0..10] := 0;
   shiftCounterDataSet[2].penultimateShiftValue.partsCurrent[0..10] := 0;
   shiftCounterDataSet[0].countPartsCurrent[0..10] := FALSE;
   shiftCounterDataSet[1].countPartsCurrent[0..10] := FALSE;
   shiftCounterDataSet[2].countPartsCurrent[0..10] := FALSE;
   shiftCounterDataSet[0].textListValue[0..10] := 0;
   shiftCounterDataSet[1].textListValue[0..10] := 0;
   shiftCounterDataSet[2].textListValue[0..10] := 0;
   shiftCounterDataSet[0..2].userInterfaceVisibility := 16#0000_0000;
   shiftCounterDataSet[0..2].resetAllExt := FALSE;
   shiftCounterDataSet[0..2].divButton := 16#00;
   shiftCounterDataSet[0..2].visibility := 16#0000_0000;
   shiftCounterOeeDataSet[0].currentShiftValue.oee[0..10] := 0.0;
   shiftCounterOeeDataSet[1].currentShiftValue.oee[0..10] := 0.0;
   shiftCounterOeeDataSet[2].currentShiftValue.oee[0..10] := 0.0;
   shiftCounterOeeDataSet[0].currentShiftValue.trend[0..10] := 0;
   shiftCounterOeeDataSet[1].currentShiftValue.trend[0..10] := 0;
   shiftCounterOeeDataSet[2].currentShiftValue.trend[0..10] := 0;
   shiftCounterOeeDataSet[0].currentShiftValue.partsTarget[0..10] := 0;
   shiftCounterOeeDataSet[1].currentShiftValue.partsTarget[0..10] := 0;
   shiftCounterOeeDataSet[2].currentShiftValue.partsTarget[0..10] := 0;
   shiftCounterOeeDataSet[0].currentShiftValue.partsCurrent[0..10] := 0;
   shiftCounterOeeDataSet[1].currentShiftValue.partsCurrent[0..10] := 0;
   shiftCounterOeeDataSet[2].currentShiftValue.partsCurrent[0..10] := 0;
   shiftCounterOeeDataSet[0].currentShiftValue.partsCurrentOk[0..10] := 0;
   shiftCounterOeeDataSet[1].currentShiftValue.partsCurrentOk[0..10] := 0;
   shiftCounterOeeDataSet[2].currentShiftValue.partsCurrentOk[0..10] := 0;
   shiftCounterOeeDataSet[0].previousShiftValue.oee[0..10] := 0.0;
   shiftCounterOeeDataSet[1].previousShiftValue.oee[0..10] := 0.0;
   shiftCounterOeeDataSet[2].previousShiftValue.oee[0..10] := 0.0;
   shiftCounterOeeDataSet[0].previousShiftValue.trend[0..10] := 0;
   shiftCounterOeeDataSet[1].previousShiftValue.trend[0..10] := 0;
   shiftCounterOeeDataSet[2].previousShiftValue.trend[0..10] := 0;
   shiftCounterOeeDataSet[0].previousShiftValue.partsTarget[0..10] := 0;
   shiftCounterOeeDataSet[1].previousShiftValue.partsTarget[0..10] := 0;
   shiftCounterOeeDataSet[2].previousShiftValue.partsTarget[0..10] := 0;
   shiftCounterOeeDataSet[0].previousShiftValue.partsCurrent[0..10] := 0;
   shiftCounterOeeDataSet[1].previousShiftValue.partsCurrent[0..10] := 0;
   shiftCounterOeeDataSet[2].previousShiftValue.partsCurrent[0..10] := 0;
   shiftCounterOeeDataSet[0].previousShiftValue.partsCurrentOk[0..10] := 0;
   shiftCounterOeeDataSet[1].previousShiftValue.partsCurrentOk[0..10] := 0;
   shiftCounterOeeDataSet[2].previousShiftValue.partsCurrentOk[0..10] := 0;
   shiftCounterOeeDataSet[0].penultimateShiftValue.oee[0..10] := 0.0;
   shiftCounterOeeDataSet[1].penultimateShiftValue.oee[0..10] := 0.0;
   shiftCounterOeeDataSet[2].penultimateShiftValue.oee[0..10] := 0.0;
   shiftCounterOeeDataSet[0].penultimateShiftValue.trend[0..10] := 0;
   shiftCounterOeeDataSet[1].penultimateShiftValue.trend[0..10] := 0;
   shiftCounterOeeDataSet[2].penultimateShiftValue.trend[0..10] := 0;
   shiftCounterOeeDataSet[0].penultimateShiftValue.partsTarget[0..10] := 0;
   shiftCounterOeeDataSet[1].penultimateShiftValue.partsTarget[0..10] := 0;
   shiftCounterOeeDataSet[2].penultimateShiftValue.partsTarget[0..10] := 0;
   shiftCounterOeeDataSet[0].penultimateShiftValue.partsCurrent[0..10] := 0;
   shiftCounterOeeDataSet[1].penultimateShiftValue.partsCurrent[0..10] := 0;
   shiftCounterOeeDataSet[2].penultimateShiftValue.partsCurrent[0..10] := 0;
   shiftCounterOeeDataSet[0].penultimateShiftValue.partsCurrentOk[0..10] := 0;
   shiftCounterOeeDataSet[1].penultimateShiftValue.partsCurrentOk[0..10] := 0;
   shiftCounterOeeDataSet[2].penultimateShiftValue.partsCurrentOk[0..10] := 0;
   shiftCounterOeeDataSet[0].countPartsCurrent[0..10] := FALSE;
   shiftCounterOeeDataSet[1].countPartsCurrent[0..10] := FALSE;
   shiftCounterOeeDataSet[2].countPartsCurrent[0..10] := FALSE;
   shiftCounterOeeDataSet[0].countPartsCurrentOk[0..10] := FALSE;
   shiftCounterOeeDataSet[1].countPartsCurrentOk[0..10] := FALSE;
   shiftCounterOeeDataSet[2].countPartsCurrentOk[0..10] := FALSE;
   shiftCounterOeeDataSet[0].textListValue[0..10] := 0;
   shiftCounterOeeDataSet[1].textListValue[0..10] := 0;
   shiftCounterOeeDataSet[2].textListValue[0..10] := 0;
   shiftCounterOeeDataSet[0..2].userInterfaceVisibility := 16#0000_0000;
   shiftCounterOeeDataSet[0..2].resetAllExt := FALSE;
   shiftCounterOeeDataSet[0..2].divButton := 16#00;
   shiftCounterOeeDataSet[0..2].visibility := 16#0000_0000;
END_DATA_BLOCK

DATA_BLOCK "ShiftInitBools"   // DB257
// stored: MemoryReserve 100
   VAR
      earlyShift : Bool := FALSE;
      lateShift : Bool := FALSE;
      nightShift : Bool := FALSE;
   END_VAR
BEGIN
END_DATA_BLOCK

DATA_BLOCK "ShiftTimesList"   // DB52
TITLE = Shifttimes / Shift times
{ DB_Accessible_From_OPC_UA := 'FALSE' }
AUTHOR : SICAR
FAMILY : Shiftmodel
// Schichtzeiten Liste / Shift times List
// stored: DBAccessibleFromOPCUA false, MemoryReserve 100
   VAR
      list { ExternalAccessible := 'False'; ExternalVisible := 'False'; ExternalWritable := 'False'} : Array[0..10] of "LSicar_typeShiftmodTime1DaySel";   // Schichtmodel Liste / Shiftmodel list
   END_VAR
BEGIN
   list[0..2].listValidFor.sunday := FALSE;
   list[3].listValidFor.sunday := TRUE;
   list[4..10].listValidFor.sunday := FALSE;
   list[0].listValidFor.monday := FALSE;
   list[1..3].listValidFor.monday := TRUE;
   list[4..10].listValidFor.monday := FALSE;
   list[0].listValidFor.tuesday := FALSE;
   list[1..3].listValidFor.tuesday := TRUE;
   list[4..10].listValidFor.tuesday := FALSE;
   list[0].listValidFor.wednesday := FALSE;
   list[1..3].listValidFor.wednesday := TRUE;
   list[4..10].listValidFor.wednesday := FALSE;
   list[0].listValidFor.thursday := FALSE;
   list[1..3].listValidFor.thursday := TRUE;
   list[4..10].listValidFor.thursday := FALSE;
   list[0].listValidFor.friday := FALSE;
   list[1].listValidFor.friday := TRUE;
   list[2].listValidFor.friday := FALSE;
   list[3].listValidFor.friday := TRUE;
   list[4..10].listValidFor.friday := FALSE;
   list[0..2].listValidFor.saturday := FALSE;
   list[3].listValidFor.saturday := TRUE;
   list[4..10].listValidFor.saturday := FALSE;
   list[0].shift[0..3].endCircuitTime := TOD#00:00:00;
   list[1].shift[0].endCircuitTime := TOD#00:00:00;
   list[1].shift[1].endCircuitTime := TOD#05:57:00;
   list[1].shift[2].endCircuitTime := TOD#13:57:00;
   list[1].shift[3].endCircuitTime := TOD#21:57:00;
   list[2].shift[0].endCircuitTime := TOD#00:00:00;
   list[2].shift[1].endCircuitTime := TOD#04:57:00;
   list[2].shift[2].endCircuitTime := TOD#14:27:00;
   list[2].shift[3].endCircuitTime := TOD#00:00:00;
   list[3].shift[0].endCircuitTime := TOD#00:00:00;
   list[3].shift[1].endCircuitTime := TOD#05:57:00;
   list[3].shift[2].endCircuitTime := TOD#14:27:00;
   list[3].shift[3].endCircuitTime := TOD#22:57:00;
   list[4].shift[0..3].endCircuitTime := TOD#00:00:00;
   list[5].shift[0..3].endCircuitTime := TOD#00:00:00;
   list[6].shift[0..3].endCircuitTime := TOD#00:00:00;
   list[7].shift[0..3].endCircuitTime := TOD#00:00:00;
   list[8].shift[0..3].endCircuitTime := TOD#00:00:00;
   list[9].shift[0..3].endCircuitTime := TOD#00:00:00;
   list[10].shift[0..3].endCircuitTime := TOD#00:00:00;
   list[0].shift[0..3].start := TOD#00:00:00;
   list[1].shift[0].start := TOD#00:00:00;
   list[1].shift[1].start := TOD#06:00:00;
   list[1].shift[2].start := TOD#14:00:00;
   list[1].shift[3].start := TOD#22:00:00;
   list[2].shift[0].start := TOD#00:00:00;
   list[2].shift[1].start := TOD#05:00:00;
   list[2].shift[2].start := TOD#14:30:00;
   list[2].shift[3].start := TOD#00:00:00;
   list[3].shift[0].start := TOD#00:00:00;
   list[3].shift[1].start := TOD#06:00:00;
   list[3].shift[2].start := TOD#14:30:00;
   list[3].shift[3].start := TOD#23:00:00;
   list[4].shift[0..3].start := TOD#00:00:00;
   list[5].shift[0..3].start := TOD#00:00:00;
   list[6].shift[0..3].start := TOD#00:00:00;
   list[7].shift[0..3].start := TOD#00:00:00;
   list[8].shift[0..3].start := TOD#00:00:00;
   list[9].shift[0..3].start := TOD#00:00:00;
   list[10].shift[0..3].start := TOD#00:00:00;
   list[0].shift[0].break[0..4].start := TOD#00:00:00;
   list[0].shift[1].break[0..4].start := TOD#00:00:00;
   list[0].shift[2].break[0..4].start := TOD#00:00:00;
   list[0].shift[3].break[0..4].start := TOD#00:00:00;
   list[1].shift[0].break[0..4].start := TOD#00:00:00;
   list[1].shift[1].break[0].start := TOD#00:00:00;
   list[1].shift[1].break[1].start := TOD#08:00:00;
   list[1].shift[1].break[2].start := TOD#10:00:00;
   list[1].shift[1].break[3].start := TOD#12:00:00;
   list[1].shift[1].break[4].start := TOD#00:00:00;
   list[1].shift[2].break[0].start := TOD#00:00:00;
   list[1].shift[2].break[1].start := TOD#16:00:00;
   list[1].shift[2].break[2].start := TOD#18:00:00;
   list[1].shift[2].break[3].start := TOD#20:00:00;
   list[1].shift[2].break[4].start := TOD#00:00:00;
   list[1].shift[3].break[0..1].start := TOD#00:00:00;
   list[1].shift[3].break[2].start := TOD#02:00:00;
   list[1].shift[3].break[3].start := TOD#04:00:00;
   list[1].shift[3].break[4].start := TOD#00:00:00;
   list[2].shift[0].break[0..4].start := TOD#00:00:00;
   list[2].shift[1].break[0].start := TOD#00:00:00;
   list[2].shift[1].break[1].start := TOD#07:00:00;
   list[2].shift[1].break[2].start := TOD#09:00:00;
   list[2].shift[1].break[3].start := TOD#11:00:00;
   list[2].shift[1].break[4].start := TOD#13:00:00;
   list[2].shift[2].break[0].start := TOD#00:00:00;
   list[2].shift[2].break[1].start := TOD#16:30:00;
   list[2].shift[2].break[2].start := TOD#18:30:00;
   list[2].shift[2].break[3].start := TOD#20:30:00;
   list[2].shift[2].break[4].start := TOD#22:00:00;
   list[2].shift[3].break[0..4].start := TOD#00:00:00;
   list[3].shift[0].break[0..4].start := TOD#00:00:00;
   list[3].shift[1].break[0].start := TOD#00:00:00;
   list[3].shift[1].break[1].start := TOD#08:00:00;
   list[3].shift[1].break[2].start := TOD#10:00:00;
   list[3].shift[1].break[3].start := TOD#11:30:00;
   list[3].shift[1].break[4].start := TOD#12:30:00;
   list[3].shift[2].break[0].start := TOD#00:00:00;
   list[3].shift[2].break[1].start := TOD#16:00:00;
   list[3].shift[2].break[2].start := TOD#18:00:00;
   list[3].shift[2].break[3].start := TOD#19:30:00;
   list[3].shift[2].break[4].start := TOD#20:30:00;
   list[3].shift[3].break[0..1].start := TOD#00:00:00;
   list[3].shift[3].break[2].start := TOD#02:00:00;
   list[3].shift[3].break[3].start := TOD#03:30:00;
   list[3].shift[3].break[4].start := TOD#04:30:00;
   list[4].shift[0].break[0..4].start := TOD#00:00:00;
   list[4].shift[1].break[0..4].start := TOD#00:00:00;
   list[4].shift[2].break[0..4].start := TOD#00:00:00;
   list[4].shift[3].break[0..4].start := TOD#00:00:00;
   list[5].shift[0].break[0..4].start := TOD#00:00:00;
   list[5].shift[1].break[0..4].start := TOD#00:00:00;
   list[5].shift[2].break[0..4].start := TOD#00:00:00;
   list[5].shift[3].break[0..4].start := TOD#00:00:00;
   list[6].shift[0].break[0..4].start := TOD#00:00:00;
   list[6].shift[1].break[0..4].start := TOD#00:00:00;
   list[6].shift[2].break[0..4].start := TOD#00:00:00;
   list[6].shift[3].break[0..4].start := TOD#00:00:00;
   list[7].shift[0].break[0..4].start := TOD#00:00:00;
   list[7].shift[1].break[0..4].start := TOD#00:00:00;
   list[7].shift[2].break[0..4].start := TOD#00:00:00;
   list[7].shift[3].break[0..4].start := TOD#00:00:00;
   list[8].shift[0].break[0..4].start := TOD#00:00:00;
   list[8].shift[1].break[0..4].start := TOD#00:00:00;
   list[8].shift[2].break[0..4].start := TOD#00:00:00;
   list[8].shift[3].break[0..4].start := TOD#00:00:00;
   list[9].shift[0].break[0..4].start := TOD#00:00:00;
   list[9].shift[1].break[0..4].start := TOD#00:00:00;
   list[9].shift[2].break[0..4].start := TOD#00:00:00;
   list[9].shift[3].break[0..4].start := TOD#00:00:00;
   list[10].shift[0].break[0..4].start := TOD#00:00:00;
   list[10].shift[1].break[0..4].start := TOD#00:00:00;
   list[10].shift[2].break[0..4].start := TOD#00:00:00;
   list[10].shift[3].break[0..4].start := TOD#00:00:00;
   list[0].shift[0].break[0..4].startCircuitTime := TOD#00:00:00;
   list[0].shift[1].break[0..4].startCircuitTime := TOD#00:00:00;
   list[0].shift[2].break[0..4].startCircuitTime := TOD#00:00:00;
   list[0].shift[3].break[0..4].startCircuitTime := TOD#00:00:00;
   list[1].shift[0].break[0..4].startCircuitTime := TOD#00:00:00;
   list[1].shift[1].break[0].startCircuitTime := TOD#00:00:00;
   list[1].shift[1].break[1].startCircuitTime := TOD#08:02:00;
   list[1].shift[1].break[2].startCircuitTime := TOD#00:00:00;
   list[1].shift[1].break[3].startCircuitTime := TOD#12:02:00;
   list[1].shift[1].break[4].startCircuitTime := TOD#00:00:00;
   list[1].shift[2].break[0].startCircuitTime := TOD#00:00:00;
   list[1].shift[2].break[1].startCircuitTime := TOD#16:02:00;
   list[1].shift[2].break[2].startCircuitTime := TOD#00:00:00;
   list[1].shift[2].break[3].startCircuitTime := TOD#20:02:00;
   list[1].shift[2].break[4].startCircuitTime := TOD#00:00:00;
   list[1].shift[3].break[0].startCircuitTime := TOD#00:00:00;
   list[1].shift[3].break[1].startCircuitTime := TOD#00:02:00;
   list[1].shift[3].break[2].startCircuitTime := TOD#00:00:00;
   list[1].shift[3].break[3].startCircuitTime := TOD#04:02:00;
   list[1].shift[3].break[4].startCircuitTime := TOD#00:00:00;
   list[2].shift[0].break[0..4].startCircuitTime := TOD#00:00:00;
   list[2].shift[1].break[0].startCircuitTime := TOD#00:00:00;
   list[2].shift[1].break[1].startCircuitTime := TOD#07:02:00;
   list[2].shift[1].break[2].startCircuitTime := TOD#00:00:00;
   list[2].shift[1].break[3].startCircuitTime := TOD#11:02:00;
   list[2].shift[1].break[4].startCircuitTime := TOD#13:02:00;
   list[2].shift[2].break[0].startCircuitTime := TOD#00:00:00;
   list[2].shift[2].break[1].startCircuitTime := TOD#16:32:00;
   list[2].shift[2].break[2].startCircuitTime := TOD#00:00:00;
   list[2].shift[2].break[3].startCircuitTime := TOD#20:32:00;
   list[2].shift[2].break[4].startCircuitTime := TOD#22:02:00;
   list[2].shift[3].break[0..4].startCircuitTime := TOD#00:00:00;
   list[3].shift[0].break[0..4].startCircuitTime := TOD#00:00:00;
   list[3].shift[1].break[0..1].startCircuitTime := TOD#00:00:00;
   list[3].shift[1].break[2].startCircuitTime := TOD#10:02:00;
   list[3].shift[1].break[3].startCircuitTime := TOD#00:00:00;
   list[3].shift[1].break[4].startCircuitTime := TOD#12:32:00;
   list[3].shift[2].break[0..1].startCircuitTime := TOD#00:00:00;
   list[3].shift[2].break[2].startCircuitTime := TOD#18:02:00;
   list[3].shift[2].break[3].startCircuitTime := TOD#00:00:00;
   list[3].shift[2].break[4].startCircuitTime := TOD#20:32:00;
   list[3].shift[3].break[0..1].startCircuitTime := TOD#00:00:00;
   list[3].shift[3].break[2].startCircuitTime := TOD#02:02:00;
   list[3].shift[3].break[3..4].startCircuitTime := TOD#00:00:00;
   list[4].shift[0].break[0..4].startCircuitTime := TOD#00:00:00;
   list[4].shift[1].break[0..4].startCircuitTime := TOD#00:00:00;
   list[4].shift[2].break[0..4].startCircuitTime := TOD#00:00:00;
   list[4].shift[3].break[0..4].startCircuitTime := TOD#00:00:00;
   list[5].shift[0].break[0..4].startCircuitTime := TOD#00:00:00;
   list[5].shift[1].break[0..4].startCircuitTime := TOD#00:00:00;
   list[5].shift[2].break[0..4].startCircuitTime := TOD#00:00:00;
   list[5].shift[3].break[0..4].startCircuitTime := TOD#00:00:00;
   list[6].shift[0].break[0..4].startCircuitTime := TOD#00:00:00;
   list[6].shift[1].break[0..4].startCircuitTime := TOD#00:00:00;
   list[6].shift[2].break[0..4].startCircuitTime := TOD#00:00:00;
   list[6].shift[3].break[0..4].startCircuitTime := TOD#00:00:00;
   list[7].shift[0].break[0..4].startCircuitTime := TOD#00:00:00;
   list[7].shift[1].break[0..4].startCircuitTime := TOD#00:00:00;
   list[7].shift[2].break[0..4].startCircuitTime := TOD#00:00:00;
   list[7].shift[3].break[0..4].startCircuitTime := TOD#00:00:00;
   list[8].shift[0].break[0..4].startCircuitTime := TOD#00:00:00;
   list[8].shift[1].break[0..4].startCircuitTime := TOD#00:00:00;
   list[8].shift[2].break[0..4].startCircuitTime := TOD#00:00:00;
   list[8].shift[3].break[0..4].startCircuitTime := TOD#00:00:00;
   list[9].shift[0].break[0..4].startCircuitTime := TOD#00:00:00;
   list[9].shift[1].break[0..4].startCircuitTime := TOD#00:00:00;
   list[9].shift[2].break[0..4].startCircuitTime := TOD#00:00:00;
   list[9].shift[3].break[0..4].startCircuitTime := TOD#00:00:00;
   list[10].shift[0].break[0..4].startCircuitTime := TOD#00:00:00;
   list[10].shift[1].break[0..4].startCircuitTime := TOD#00:00:00;
   list[10].shift[2].break[0..4].startCircuitTime := TOD#00:00:00;
   list[10].shift[3].break[0..4].startCircuitTime := TOD#00:00:00;
   list[0].shift[0].break[0..4].endCircuitTime := TOD#00:00:00;
   list[0].shift[1].break[0..4].endCircuitTime := TOD#00:00:00;
   list[0].shift[2].break[0..4].endCircuitTime := TOD#00:00:00;
   list[0].shift[3].break[0..4].endCircuitTime := TOD#00:00:00;
   list[1].shift[0].break[0..4].endCircuitTime := TOD#00:00:00;
   list[1].shift[1].break[0].endCircuitTime := TOD#00:00:00;
   list[1].shift[1].break[1].endCircuitTime := TOD#08:13:00;
   list[1].shift[1].break[2].endCircuitTime := TOD#00:00:00;
   list[1].shift[1].break[3].endCircuitTime := TOD#12:13:00;
   list[1].shift[1].break[4].endCircuitTime := TOD#00:00:00;
   list[1].shift[2].break[0].endCircuitTime := TOD#00:00:00;
   list[1].shift[2].break[1].endCircuitTime := TOD#16:13:00;
   list[1].shift[2].break[2].endCircuitTime := TOD#00:00:00;
   list[1].shift[2].break[3].endCircuitTime := TOD#20:13:00;
   list[1].shift[2].break[4].endCircuitTime := TOD#00:00:00;
   list[1].shift[3].break[0].endCircuitTime := TOD#00:00:00;
   list[1].shift[3].break[1].endCircuitTime := TOD#00:13:00;
   list[1].shift[3].break[2].endCircuitTime := TOD#00:00:00;
   list[1].shift[3].break[3].endCircuitTime := TOD#04:13:00;
   list[1].shift[3].break[4].endCircuitTime := TOD#00:00:00;
   list[2].shift[0].break[0..4].endCircuitTime := TOD#00:00:00;
   list[2].shift[1].break[0].endCircuitTime := TOD#00:00:00;
   list[2].shift[1].break[1].endCircuitTime := TOD#07:13:00;
   list[2].shift[1].break[2].endCircuitTime := TOD#00:00:00;
   list[2].shift[1].break[3].endCircuitTime := TOD#11:13:00;
   list[2].shift[1].break[4].endCircuitTime := TOD#13:13:00;
   list[2].shift[2].break[0].endCircuitTime := TOD#00:00:00;
   list[2].shift[2].break[1].endCircuitTime := TOD#16:43:00;
   list[2].shift[2].break[2].endCircuitTime := TOD#00:00:00;
   list[2].shift[2].break[3].endCircuitTime := TOD#20:43:00;
   list[2].shift[2].break[4].endCircuitTime := TOD#22:13:00;
   list[2].shift[3].break[0..4].endCircuitTime := TOD#00:00:00;
   list[3].shift[0].break[0..4].endCircuitTime := TOD#00:00:00;
   list[3].shift[1].break[0..1].endCircuitTime := TOD#00:00:00;
   list[3].shift[1].break[2].endCircuitTime := TOD#10:13:00;
   list[3].shift[1].break[3].endCircuitTime := TOD#00:00:00;
   list[3].shift[1].break[4].endCircuitTime := TOD#12:43:00;
   list[3].shift[2].break[0..1].endCircuitTime := TOD#00:00:00;
   list[3].shift[2].break[2].endCircuitTime := TOD#18:13:00;
   list[3].shift[2].break[3].endCircuitTime := TOD#00:00:00;
   list[3].shift[2].break[4].endCircuitTime := TOD#20:43:00;
   list[3].shift[3].break[0..1].endCircuitTime := TOD#00:00:00;
   list[3].shift[3].break[2].endCircuitTime := TOD#02:13:00;
   list[3].shift[3].break[3..4].endCircuitTime := TOD#00:00:00;
   list[4].shift[0].break[0..4].endCircuitTime := TOD#00:00:00;
   list[4].shift[1].break[0..4].endCircuitTime := TOD#00:00:00;
   list[4].shift[2].break[0..4].endCircuitTime := TOD#00:00:00;
   list[4].shift[3].break[0..4].endCircuitTime := TOD#00:00:00;
   list[5].shift[0].break[0..4].endCircuitTime := TOD#00:00:00;
   list[5].shift[1].break[0..4].endCircuitTime := TOD#00:00:00;
   list[5].shift[2].break[0..4].endCircuitTime := TOD#00:00:00;
   list[5].shift[3].break[0..4].endCircuitTime := TOD#00:00:00;
   list[6].shift[0].break[0..4].endCircuitTime := TOD#00:00:00;
   list[6].shift[1].break[0..4].endCircuitTime := TOD#00:00:00;
   list[6].shift[2].break[0..4].endCircuitTime := TOD#00:00:00;
   list[6].shift[3].break[0..4].endCircuitTime := TOD#00:00:00;
   list[7].shift[0].break[0..4].endCircuitTime := TOD#00:00:00;
   list[7].shift[1].break[0..4].endCircuitTime := TOD#00:00:00;
   list[7].shift[2].break[0..4].endCircuitTime := TOD#00:00:00;
   list[7].shift[3].break[0..4].endCircuitTime := TOD#00:00:00;
   list[8].shift[0].break[0..4].endCircuitTime := TOD#00:00:00;
   list[8].shift[1].break[0..4].endCircuitTime := TOD#00:00:00;
   list[8].shift[2].break[0..4].endCircuitTime := TOD#00:00:00;
   list[8].shift[3].break[0..4].endCircuitTime := TOD#00:00:00;
   list[9].shift[0].break[0..4].endCircuitTime := TOD#00:00:00;
   list[9].shift[1].break[0..4].endCircuitTime := TOD#00:00:00;
   list[9].shift[2].break[0..4].endCircuitTime := TOD#00:00:00;
   list[9].shift[3].break[0..4].endCircuitTime := TOD#00:00:00;
   list[10].shift[0].break[0..4].endCircuitTime := TOD#00:00:00;
   list[10].shift[1].break[0..4].endCircuitTime := TOD#00:00:00;
   list[10].shift[2].break[0..4].endCircuitTime := TOD#00:00:00;
   list[10].shift[3].break[0..4].endCircuitTime := TOD#00:00:00;
   list[0].shift[0].break[0..4].end := TOD#00:00:00;
   list[0].shift[1].break[0..4].end := TOD#00:00:00;
   list[0].shift[2].break[0..4].end := TOD#00:00:00;
   list[0].shift[3].break[0..4].end := TOD#00:00:00;
   list[1].shift[0].break[0..4].end := TOD#00:00:00;
   list[1].shift[1].break[0].end := TOD#00:00:00;
   list[1].shift[1].break[1].end := TOD#08:15:00;
   list[1].shift[1].break[2].end := TOD#10:10:00;
   list[1].shift[1].break[3].end := TOD#12:15:00;
   list[1].shift[1].break[4].end := TOD#00:00:00;
   list[1].shift[2].break[0].end := TOD#00:00:00;
   list[1].shift[2].break[1].end := TOD#16:15:00;
   list[1].shift[2].break[2].end := TOD#18:10:00;
   list[1].shift[2].break[3].end := TOD#20:15:00;
   list[1].shift[2].break[4].end := TOD#00:00:00;
   list[1].shift[3].break[0].end := TOD#00:00:00;
   list[1].shift[3].break[1].end := TOD#00:15:00;
   list[1].shift[3].break[2].end := TOD#02:10:00;
   list[1].shift[3].break[3].end := TOD#04:15:00;
   list[1].shift[3].break[4].end := TOD#00:00:00;
   list[2].shift[0].break[0..4].end := TOD#00:00:00;
   list[2].shift[1].break[0].end := TOD#00:00:00;
   list[2].shift[1].break[1].end := TOD#07:15:00;
   list[2].shift[1].break[2].end := TOD#09:10:00;
   list[2].shift[1].break[3].end := TOD#11:15:00;
   list[2].shift[1].break[4].end := TOD#13:15:00;
   list[2].shift[2].break[0].end := TOD#00:00:00;
   list[2].shift[2].break[1].end := TOD#16:45:00;
   list[2].shift[2].break[2].end := TOD#18:40:00;
   list[2].shift[2].break[3].end := TOD#20:45:00;
   list[2].shift[2].break[4].end := TOD#22:15:00;
   list[2].shift[3].break[0..4].end := TOD#00:00:00;
   list[3].shift[0].break[0..4].end := TOD#00:00:00;
   list[3].shift[1].break[0].end := TOD#00:00:00;
   list[3].shift[1].break[1].end := TOD#08:10:00;
   list[3].shift[1].break[2].end := TOD#10:15:00;
   list[3].shift[1].break[3].end := TOD#11:40:00;
   list[3].shift[1].break[4].end := TOD#12:45:00;
   list[3].shift[2].break[0].end := TOD#00:00:00;
   list[3].shift[2].break[1].end := TOD#16:10:00;
   list[3].shift[2].break[2].end := TOD#18:15:00;
   list[3].shift[2].break[3].end := TOD#19:40:00;
   list[3].shift[2].break[4].end := TOD#20:45:00;
   list[3].shift[3].break[0].end := TOD#00:00:00;
   list[3].shift[3].break[1].end := TOD#00:10:00;
   list[3].shift[3].break[2].end := TOD#02:15:00;
   list[3].shift[3].break[3].end := TOD#03:40:00;
   list[3].shift[3].break[4].end := TOD#04:45:00;
   list[4].shift[0].break[0..4].end := TOD#00:00:00;
   list[4].shift[1].break[0..4].end := TOD#00:00:00;
   list[4].shift[2].break[0..4].end := TOD#00:00:00;
   list[4].shift[3].break[0..4].end := TOD#00:00:00;
   list[5].shift[0].break[0..4].end := TOD#00:00:00;
   list[5].shift[1].break[0..4].end := TOD#00:00:00;
   list[5].shift[2].break[0..4].end := TOD#00:00:00;
   list[5].shift[3].break[0..4].end := TOD#00:00:00;
   list[6].shift[0].break[0..4].end := TOD#00:00:00;
   list[6].shift[1].break[0..4].end := TOD#00:00:00;
   list[6].shift[2].break[0..4].end := TOD#00:00:00;
   list[6].shift[3].break[0..4].end := TOD#00:00:00;
   list[7].shift[0].break[0..4].end := TOD#00:00:00;
   list[7].shift[1].break[0..4].end := TOD#00:00:00;
   list[7].shift[2].break[0..4].end := TOD#00:00:00;
   list[7].shift[3].break[0..4].end := TOD#00:00:00;
   list[8].shift[0].break[0..4].end := TOD#00:00:00;
   list[8].shift[1].break[0..4].end := TOD#00:00:00;
   list[8].shift[2].break[0..4].end := TOD#00:00:00;
   list[8].shift[3].break[0..4].end := TOD#00:00:00;
   list[9].shift[0].break[0..4].end := TOD#00:00:00;
   list[9].shift[1].break[0..4].end := TOD#00:00:00;
   list[9].shift[2].break[0..4].end := TOD#00:00:00;
   list[9].shift[3].break[0..4].end := TOD#00:00:00;
   list[10].shift[0].break[0..4].end := TOD#00:00:00;
   list[10].shift[1].break[0..4].end := TOD#00:00:00;
   list[10].shift[2].break[0..4].end := TOD#00:00:00;
   list[10].shift[3].break[0..4].end := TOD#00:00:00;
   list[0].shift[0..3].end := TOD#00:00:00;
   list[1].shift[0].end := TOD#00:00:00;
   list[1].shift[1].end := TOD#13:30:00;
   list[1].shift[2].end := TOD#21:30:00;
   list[1].shift[3].end := TOD#05:30:00;
   list[2].shift[0].end := TOD#00:00:00;
   list[2].shift[1].end := TOD#14:00:00;
   list[2].shift[2].end := TOD#23:30:00;
   list[2].shift[3].end := TOD#00:00:00;
   list[3].shift[0].end := TOD#00:00:00;
   list[3].shift[1].end := TOD#13:30:00;
   list[3].shift[2].end := TOD#21:30:00;
   list[3].shift[3].end := TOD#05:30:00;
   list[4].shift[0..3].end := TOD#00:00:00;
   list[5].shift[0..3].end := TOD#00:00:00;
   list[6].shift[0..3].end := TOD#00:00:00;
   list[7].shift[0..3].end := TOD#00:00:00;
   list[8].shift[0..3].end := TOD#00:00:00;
   list[9].shift[0..3].end := TOD#00:00:00;
   list[10].shift[0..3].end := TOD#00:00:00;
   list[0].shift[0..3].startCircuitTime := TOD#00:00:00;
   list[1].shift[0].startCircuitTime := TOD#00:00:00;
   list[1].shift[1].startCircuitTime := TOD#13:33:00;
   list[1].shift[2].startCircuitTime := TOD#21:33:00;
   list[1].shift[3].startCircuitTime := TOD#05:33:00;
   list[2].shift[0].startCircuitTime := TOD#00:00:00;
   list[2].shift[1].startCircuitTime := TOD#14:03:00;
   list[2].shift[2].startCircuitTime := TOD#23:33:00;
   list[2].shift[3].startCircuitTime := TOD#00:00:00;
   list[3].shift[0].startCircuitTime := TOD#00:00:00;
   list[3].shift[1].startCircuitTime := TOD#13:33:00;
   list[3].shift[2].startCircuitTime := TOD#21:33:00;
   list[3].shift[3].startCircuitTime := TOD#05:33:00;
   list[4].shift[0..3].startCircuitTime := TOD#00:00:00;
   list[5].shift[0..3].startCircuitTime := TOD#00:00:00;
   list[6].shift[0..3].startCircuitTime := TOD#00:00:00;
   list[7].shift[0..3].startCircuitTime := TOD#00:00:00;
   list[8].shift[0..3].startCircuitTime := TOD#00:00:00;
   list[9].shift[0..3].startCircuitTime := TOD#00:00:00;
   list[10].shift[0..3].startCircuitTime := TOD#00:00:00;
END_DATA_BLOCK

DATA_BLOCK "Settings"   // DB6
{ DB_Accessible_From_OPC_UA := 'FALSE' }
// stored: DBAccessibleFromOPCUA false, DBAccessibleFromWebserver false, MemoryReserve 100
   VAR
      diagPlc : "LAF_typePlcDiag";   // HMI Schnittstelle PLC Diagnose / HMI interface PLC diag
      checksum : "LAF_typeChecksum";   // HMI Schnittstelle PLCChecksum / HMI interface PLCChecksum
      diagMemCard : "LAF_typeMemCardDiag";   // HMI Schnittstelle SMCDiag / HMI interface SMCDiag
      cycleTimes : "LSicar_typeGlobalRuntime";
      setLocalPlcTime : "LAF_typeSetPlcTime";
      ITConnection : Bool := FALSE;   // Provides a visual representation of the connection with the IT systems.
   END_VAR
BEGIN
   diagPlc.manualReadAll := FALSE;
   diagPlc.blockBusyAfterRestart := FALSE;
   diagPlc.im0Data.Manufacturer_ID := 42;
   diagPlc.im0Data.Order_ID := '6ES7 518-3UT10-0AB0 ';
   diagPlc.im0Data.Serial_Number := 'S C-T4A0RVHM2025';
   diagPlc.im0Data.Hardware_Revision := 1;
   diagPlc.im0Data.Software_Revision."Type" := 'V';
   diagPlc.im0Data.Software_Revision.Functional := 4;
   diagPlc.im0Data.Software_Revision.Bugfix := 0;
   diagPlc.im0Data.Software_Revision.Internal := 0;
   diagPlc.im0Data.Revision_Counter := 0;
   diagPlc.im0Data.Profile_ID := 0;
   diagPlc.im0Data.Profile_Specific_Type := 0;
   diagPlc.im0Data.IM_Version := 16#0101;
   diagPlc.im0Data.IM_Supported := 16#000E;
   diagPlc.im1PlantDesignLocIdent := '                                                      ';
   diagPlc.im1PlantDesignation := '                                ';
   diagPlc.im1LocIdent := '                      ';
   diagPlc.im2InstallationDate := '2025-02-24 16:59';
   diagPlc.im3AdditionalInfo := '                                                      ';
   diagPlc.addressMac[0] := 16#30;
   diagPlc.addressMac[1] := 16#B8;
   diagPlc.addressMac[2] := 16#51;
   diagPlc.addressMac[3] := 16#66;
   diagPlc.addressMac[4] := 16#CF;
   diagPlc.addressMac[5] := 16#66;
   diagPlc.addressIpV4[0] := 192;
   diagPlc.addressIpV4[1] := 168;
   diagPlc.addressIpV4[2] := 200;
   diagPlc.addressIpV4[3] := 51;
   diagPlc.addressSubnet[0..2] := 255;
   diagPlc.addressSubnet[3] := 0;
   diagPlc.im0SwRev := 'V';
   checksum.checksumStandard := 'E4AA23DFFDEEA866';
   checksum.checksumStandardOld := 'E4AA23DFFDEEA866';
   checksum.checksumSafety := '0A6CEC4B00000000';
   checksum.checksumSafetyOld := '0A6CEC4B00000000';
   checksum.checksumTextlists := '676DC45055902179';
   checksum.checksumTextlistsOld := '676DC45055902179';
   checksum.dateTimeStandardModified := DT#2026-01-06-00:09:42.545;
   checksum.dateTimeSafetyModified := DT#2026-01-06-00:09:42.545;
   checksum.dateTimeTextlistModified := DT#2026-01-06-00:09:42.545;
   checksum.standardModified := FALSE;
   checksum.safetyModified := FALSE;
   checksum.textlistsModified := FALSE;
   checksum.summaryModified := FALSE;
   checksum.updateValuesOld := FALSE;
   diagMemCard.alarmWarnInfo := 16#00;
   diagMemCard.manualUpdate := FALSE;
   diagMemCard.memorySpaceKbyte := 31151664;
   diagMemCard.assignedMemorySpaceKbyte := 68208;
   diagMemCard.assignedMemorySpace := 0;
   diagMemCard.usedLifetime := 0;
   diagMemCard.paraLifetime := 80;
   diagMemCard.warningFromMemorySpace := 81;
   diagMemCard.alarmFromMemorySpace := 95;
   cycleTimes.prevCycle := 3;
   cycleTimes.reset := FALSE;
   cycleTimes.maxCycle := 5;
   cycleTimes.minCycle := 2;
   cycleTimes.maxCycleRuntime := 100;
   cycleTimes.minCycleRuntime := 1;
   cycleTimes.maxCommRuntime := 0;
   setLocalPlcTime.newDateAndTime := DT#1990-01-01-00:00:00;
   setLocalPlcTime.daylightSavingTime := FALSE;
   setLocalPlcTime.apply := FALSE;
END_DATA_BLOCK

DATA_BLOCK "HMI_Interface_Parameter"   // DB262
// stored: Access Published, MemoryReserve 100
   VAR RETAIN
      ProcessUnitSelect : Int := 4;   // 1. Anode Reel Cut, 2. Cathode Reel Cut, 3. Stacking#1, 4.Stacking#2, 5. Inspection
   END_VAR
   VAR
      Recipe : "HMI_IF_Parameter_LIstRecipe_Interface";
      RecipeButton : "HMI_IF_Parameter_Save Button_UDT";
   END_VAR
   VAR RETAIN
      "Default Recipe" : "HMI_IF_Parameter_Recipe_Electrod_Interface";
      "Reelcut Recipe" { S7_SetPoint := 'True'} : "HMI_IF_Parameter_Recipe_Electrod_Reelcut_Interface";
      Parameter_Image : Array[0..17] of "HMI_IF_Parameter_Parameter_UDT";
      Parameter_Text : Array[0..154] of "HMI_IF_Parameter_Parameter_UDT";
      "Save Button" : "HMI_IF_Parameter_Save Button_UDT";
   END_VAR
   VAR
      "Save Button Old" { S7_SetPoint := 'True'} : "HMI_IF_Parameter_Save Button_UDT";
   END_VAR
   VAR RETAIN
      FATModeSelect : "LER_TypeFATMode_ModeSelect";
      FATModeInterface { S7_SetPoint := 'True'} : "LER_TypeFATModeInterface";
      VisionProgramNum : DWord;
   END_VAR
   VAR
      TempNull : Bool;
      TeachingPosIndex : SInt;
   END_VAR
   VAR RETAIN
      TeachingPosInterface : Array[0..48] of "LER_TypeTeachingPosInterface";
   END_VAR
   VAR
      PulseBit { ExternalAccessible := 'False'; ExternalVisible := 'False'; ExternalWritable := 'False'} : Array[0..99] of Bool;
   END_VAR
   VAR RETAIN
      Softcam : Array[0..48] of "LER_typeSoftCamRelation";
   END_VAR
   VAR
      SoftcamIndex : SInt;
   END_VAR
BEGIN
   // Parameter_Text[0] : CPM
   // Parameter_Text[2] : CellCount
   // Parameter_Text[6] : SleepModeActivationTime
   // Parameter_Text[7] : DeepSleepModeActivationTime
   // Parameter_Text[9] : Setpoint
   // Parameter_Text[10] : Kp
   // Parameter_Text[11] : Ki
   // Parameter_Text[13] : Pos1FinalRollerXFwdOutputCam
   // Parameter_Text[14] : Pos1FinalRollerXBwdOutputCam
   // Parameter_Text[15] : Pos1FinalRollerXStackTableDownOutputCam
   // Parameter_Text[16] : Pos1FinalRollerXStackAnodeVisionOutputCam
   // Parameter_Text[17] : Pos1FinalRollerXStackCathodeVisionOutputCam
   // Parameter_Text[18] : Pos1AnodePnPX1FwdOutputCam
   // Parameter_Text[19] : Pos1AnodePnPX1BwdOutputCam
   // Parameter_Text[20] : Pos1AnodePnPX1ReelCutDataDeleteOffOutputCam
   // Parameter_Text[21] : Pos1AnodePnPX2FwdOutputCam
   // Parameter_Text[22] : Pos1AnodePnPX2BwdOutputCam
   // Parameter_Text[23] : Pos1AnodePnPZ1Down1OutputCam
   // Parameter_Text[24] : Pos1AnodePnPZ1Up1OutputCam
   // Parameter_Text[25] : Pos1AnodePnPZ2Down1OutputCam
   // Parameter_Text[26] : Pos1AnodePnPZ2Up1OutputCam
   // Parameter_Text[27] : Pos1AnodePnPZ1Down2OutputCam
   // Parameter_Text[28] : Pos1AnodePnPZ1Up2OutputCam
   // Parameter_Text[29] : Pos1AnodePnPZ2Down2OutputCam
   // Parameter_Text[30] : Pos1AnodePnPZ2Up2OutputCam
   // Parameter_Text[31] : Pos1AnodePnPZ1SuctionOnOutputCam
   // Parameter_Text[32] : Pos1AnodePnPZ1SuctionOffOutputCam
   // Parameter_Text[33] : Pos1AnodePnPZ1ReelCutBlowOutputCam
   // Parameter_Text[34] : Pos1AnodePnPZ1ReelCutDataDeleteOnOutputCam
   // Parameter_Text[35] : Pos1AnodePnPZ1AlignVisionOutputCam
   // Parameter_Text[36] : Pos1AnodePnPZ2SuctionOnOutputCam
   // Parameter_Text[37] : Pos1AnodePnPZ2SuctionOffOutputCam
   // Parameter_Text[38] : Pos1AnodeAlignSuctionOnOutputCam
   // Parameter_Text[39] : Pos1AnodeAlignSuctionOffOutputCam
   // Parameter_Text[40] : Pos1CathodePnPX1FwdOutputCam
   // Parameter_Text[41] : Pos1CathodePnPX1BwdOutputCam
   // Parameter_Text[42] : Pos1CathodePnPX1ReelCutDataDeleteOffOutputCam
   // Parameter_Text[43] : Pos1CathodePnPX2FwdOutputCam
   // Parameter_Text[44] : Pos1CathodePnPX2BwdOutputCam
   // Parameter_Text[45] : Pos1CathodePnPZ1Down1OutputCam
   // Parameter_Text[46] : Pos1CathodePnPZ1Up1OutputCam
   // Parameter_Text[47] : Pos1CathodePnPZ2Down1OutputCam
   // Parameter_Text[48] : Pos1CathodePnPZ2Up1OutputCam
   // Parameter_Text[49] : Pos1CathodePnPZ1Down2OutputCam
   // Parameter_Text[50] : Pos1CathodePnPZ1Up2OutputCam
   // Parameter_Text[51] : Pos1CathodePnPZ2Down2OutputCam
   // Parameter_Text[52] : Pos1CathodePnPZ2Up2OutputCam
   // Parameter_Text[53] : Pos1CathodePnPZ1SuctionOnOutputCam
   // Parameter_Text[54] : Pos1CathodePnPZ1SuctionOffOutputCam
   // Parameter_Text[55] : Pos1CathodePnPZ1ReelCutBlowOutputCam
   // Parameter_Text[56] : Pos1CathodePnPZ1ReelCutDataDeleteOnOutputCam
   // Parameter_Text[57] : Pos1CathodePnPZ1AlignVisionOutputCam
   // Parameter_Text[58] : Pos1CathodePnPZ2SuctionOnOutputCam
   // Parameter_Text[59] : Pos1CathodePnPZ2SuctionOffOutputCam
   // Parameter_Text[60] : Pos1CathodeAlignSuctionOnOutputCam
   // Parameter_Text[61] : Pos1CathodeAlignSuctionOffOutputCam
   // Parameter_Text[62] : Pos2FinalRollerXFwdOutputCam
   // Parameter_Text[63] : Pos2FinalRollerXBwdOutputCam
   // Parameter_Text[64] : Pos2FinalRollerXStackTableDownOutputCam
   // Parameter_Text[65] : Pos2FinalRollerXStackAnodeVisionOutputCam
   // Parameter_Text[66] : Pos2FinalRollerXStackCathodeVisionOutputCam
   // Parameter_Text[67] : Pos2AnodePnPX1FwdOutputCam
   // Parameter_Text[68] : Pos2AnodePnPX1BwdOutputCam
   // Parameter_Text[69] : Pos2AnodePnPX1ReelCutDataDeleteOffOutputCam
   // Parameter_Text[70] : Pos2AnodePnPX2FwdOutputCam
   // Parameter_Text[71] : Pos2AnodePnPX2BwdOutputCam
   // Parameter_Text[72] : Pos2AnodePnPZ1Down1OutputCam
   // Parameter_Text[73] : Pos2AnodePnPZ1Up1OutputCam
   // Parameter_Text[74] : Pos2AnodePnPZ2Down1OutputCam
   // Parameter_Text[75] : Pos2AnodePnPZ2Up1OutputCam
   // Parameter_Text[76] : Pos2AnodePnPZ1Down2OutputCam
   // Parameter_Text[77] : Pos2AnodePnPZ1Up2OutputCam
   // Parameter_Text[78] : Pos2AnodePnPZ2Down2OutputCam
   // Parameter_Text[79] : Pos2AnodePnPZ2Up2OutputCam
   // Parameter_Text[80] : Pos2AnodePnPZ1SuctionOnOutputCam
   // Parameter_Text[81] : Pos2AnodePnPZ1SuctionOffOutputCam
   // Parameter_Text[82] : Pos2AnodePnPZ1ReelCutBlowOutputCam
   // Parameter_Text[83] : Pos2AnodePnPZ1ReelCutDataDeleteOnOutputCam
   // Parameter_Text[84] : Pos2AnodePnPZ1AlignVisionOutputCam
   // Parameter_Text[85] : Pos2AnodePnPZ2SuctionOnOutputCam
   // Parameter_Text[86] : Pos2AnodePnPZ2SuctionOffOutputCam
   // Parameter_Text[87] : Pos2AnodeAlignSuctionOnOutputCam
   // Parameter_Text[88] : Pos2AnodeAlignSuctionOffOutputCam
   // Parameter_Text[89] : Pos2CathodePnPX1FwdOutputCam
   // Parameter_Text[90] : Pos2CathodePnPX1BwdOutputCam
   // Parameter_Text[91] : Pos2CathodePnPX1ReelCutDataDeleteOffOutputCam
   // Parameter_Text[92] : Pos2CathodePnPX2FwdOutputCam
   // Parameter_Text[93] : Pos2CathodePnPX2BwdOutputCam
   // Parameter_Text[94] : Pos2CathodePnPZ1Down1OutputCam
   // Parameter_Text[95] : Pos2CathodePnPZ1Up1OutputCam
   // Parameter_Text[96] : Pos2CathodePnPZ2Down1OutputCam
   // Parameter_Text[97] : Pos2CathodePnPZ2Up1OutputCam
   // Parameter_Text[98] : Pos2CathodePnPZ1Down2OutputCam
   // Parameter_Text[99] : Pos2CathodePnPZ1Up2OutputCam
   // Parameter_Text[100] : Pos2CathodePnPZ2Down2OutputCam
   // Parameter_Text[101] : Pos2CathodePnPZ2Up2OutputCam
   // Parameter_Text[102] : Pos2CathodePnPZ1SuctionOnOutputCam
   // Parameter_Text[103] : Pos2CathodePnPZ1SuctionOffOutputCam
   // Parameter_Text[104] : Pos2CathodePnPZ1ReelCutBlowOutputCam
   // Parameter_Text[105] : Pos2CathodePnPZ1ReelCutDataDeleteOnOutputCam
   // Parameter_Text[106] : Pos2CathodePnPZ1AlignVisionOutputCam
   // Parameter_Text[107] : Pos2CathodePnPZ2SuctionOnOutputCam
   // Parameter_Text[108] : Pos2CathodePnPZ2SuctionOffOutputCam
   // Parameter_Text[109] : Pos2CathodeAlignSuctionOnOutputCam
   // Parameter_Text[110] : Pos2CathodeAlignSuctionOffOutputCam
   // Parameter_Text[111] : StageHeight
   // Parameter_Text[112] : StageGap
   // Parameter_Text[113] : FinalRollerStart
   // Parameter_Text[114] : FinalRollerEnd
   // Parameter_Text[115] : PnPXStart
   // Parameter_Text[116] : PnPXEnd
   // Parameter_Text[117] : PnPZDownStart
   // Parameter_Text[118] : PnPZDownEnd
   // Parameter_Text[119] : PnPZUpStart
   // Parameter_Text[120] : PnPZUpEnd
   // Parameter_Text[121] : MandrelBwdStart
   // Parameter_Text[122] : MandrelBwdEnd
   // Parameter_Text[123] : MandrelFwdStart
   // Parameter_Text[124] : MandrelFwdEnd
   // Parameter_Text[125] : MandrelUpStart1
   // Parameter_Text[126] : MandrelUpEnd1
   // Parameter_Text[127] : MandrelUpStart2
   // Parameter_Text[128] : MandrelUpEnd2
   // Parameter_Text[129] : MandrelDownStart
   // Parameter_Text[130] : MandrelDownEnd
   // Parameter_Text[131] : MandrelYTerm
   // Parameter_Text[132] : MandrelZTerm
   // Parameter_Text[133] : MandrelBwdOffset
   // Parameter_Text[134] : MandrelFwdOffset
   // Parameter_Text[135] : FinalRollerStart
   // Parameter_Text[136] : FinalRollerEnd
   // Parameter_Text[137] : PnPXStart
   // Parameter_Text[138] : PnPXEnd
   // Parameter_Text[139] : PnPZDownStart
   // Parameter_Text[140] : PnPZDownEnd
   // Parameter_Text[141] : PnPZUpStart
   // Parameter_Text[142] : PnPZUpEnd
   // Parameter_Text[143] : MandrelBwdStart
   // Parameter_Text[144] : MandrelBwdEnd
   // Parameter_Text[145] : MandrelFwdStart
   // Parameter_Text[146] : MandrelFwdEnd
   // Parameter_Text[147] : MandrelUpStart1
   // Parameter_Text[148] : MandrelUpEnd1
   // Parameter_Text[149] : MandrelUpStart2
   // Parameter_Text[150] : MandrelUpEnd2
   // Parameter_Text[151] : MandrelDownStart
   // Parameter_Text[152] : MandrelDownEnd
   // Parameter_Text[153] : FinalRollerBwdPos
   // Parameter_Text[154] : FinalRollerFwdPos
END_DATA_BLOCK

DATA_BLOCK "RecipeParameter"   // DB115
// stored: Access Published, MemoryReserve 100
   VAR
      SelectdRecipeTypeID : Int;
      SelectdRecipeID : Int;
      CurrentRecipeName : WString;
      CurrentRecipeID : Int;
      GetParameterSetName : Int;
      ParametersSV : "HMI_IF_Parameter_ListRecipe_UDT";
      ParametersPV : "HMI_IF_Parameter_ListRecipe_UDT";
   END_VAR
BEGIN
END_DATA_BLOCK

DATA_BLOCK "ManualOperationControl_CITIEm1"   // DB447
// stored: MemoryReserve 100
   VAR
      manualOperationEm { ExternalAccessible := 'False'; ExternalVisible := 'False'; ExternalWritable := 'False'} : "LAF_typeManEm";
      manualOperationEmArea { ExternalAccessible := 'False'; ExternalVisible := 'False'; ExternalWritable := 'False'} : Array[1..5] of "LAF_typeManOperationArea";
      manualOperationCms { ExternalAccessible := 'False'; ExternalVisible := 'False'; ExternalWritable := 'False'} : Array[1..41] of "LAF_typeManOperation";
   END_VAR
BEGIN
   manualOperationEm.equipmentModuleNum := 1080;
END_DATA_BLOCK

